FUNCTION_BLOCK UN_Machine EXTENDS FB_UN_PackML_Base
VAR_INPUT
END_VAR
VAR_OUTPUT
END_VAR
VAR
	// HMI
	s_stHmi : ST_UN_Machine_Hmi;
	
END_VAR

SUPER^();

METHOD PROTECTED _m_Alarms
SUPER^._m_Alarms();
END_METHOD

METHOD PROTECTED _m_Hmi
SUPER^._m_Hmi();

s_stHmi.fbHmiAlarmCollector(i_itfAlarmCollector := s_fbAlarmCollector);
END_METHOD

METHOD PROTECTED _m_Logic
SUPER^._m_Logic();

_m_Hmi();
END_METHOD

METHOD PROTECTED _m_Modules
SUPER^._m_Modules();

GVL_Modules.g_emInfeedConveyor(
	i_bReqEnable					:= TRUE, 
	i_bReqReset						:= s_fbAlarmCollector.q_bReqReset, 
	i_bStaSafetyOk					:= TRUE, 
	i_bReqSimulation				:= p_bStaSimulation, 
	i_itfPackML_Parent				:= s_fbPackML, 
	i_itfAlarmCollector_Parent		:= s_fbAlarmCollector, 
	q_stStaPackML					=> );
END_METHOD

METHOD PUBLIC m_Main
SUPER^.m_Main();
END_METHOD

END_FUNCTION_BLOCK

(* stored: Version 1.1.0.1, ProductVersion 3.1.4026.13
   POU UN_Machine: Id {21e30d72-cc39-422e-8114-15c7abc2b847}, SpecialFunc None
   Folder Basic: Id {e89104c0-d33f-460a-aaf2-8953cfda25ab}
   Method _m_Alarms: Id {8fa8464a-636c-46ee-9f13-6e7927953bcd}
   Method _m_Hmi: Id {e2052703-323d-40e8-9f21-012122f38ffa}
   Method _m_Logic: Id {b95711e4-a3f3-4e91-9f55-7c0e3689d897}
   Method _m_Modules: Id {c15e282d-b76d-440b-8236-902bb4c31743}
   Method m_Main: Id {5738c138-41a1-473c-badd-a5f9691bbc49} *)
